(* PLC project Untitled1, Beckhoff Automation GmbH TwinCAT PLC Control 3.5.13.20 *)
(* stored: creationDateTime 2022-07-20T15:23:05.6676109, modificationDateTime 2022-07-20T15:23:05.6676109 *)

TYPE ST_FirmerPvInverter_Data : STRUCT
  eOperatingState : eFirmerOperatingState;  (* Operating State *)
  eEvent1 : eFirmerEvent;  (* Eventfield *)
  eVendorEvent1 : eFirmerVendorEvent1;  (* Vendor Event 1 *)
  eVendorEvent2 : eFirmerVendorEvent2;  (* Vendor Event 2 *)
  eVendorEvent3 : eFirmerVendorEvent3;  (* Vendor Event 3 *)
  rTotalMPPTPower : REAL;  (* Total DC Power in kW from the MPPT *)
  rCabinetTemp : REAL;  (* Cabinet Temperature *)
  rHeatSinkTemp : REAL;  (* Heat Sink Temperature *)
  arrMPPTPower : ARRAY[1..6] OF REAL;  (* Each MPPT DC Power in kW (Max 6 MPPT) *)
END_STRUCT;
END_TYPE
